(* PLC project Tc3_EventLogger.ipArguments Demo, tc3-libraries-kb TwinCAT 3.1 *)
(* stored: creationDateTime 2026-05-11T01:00:00, modificationDateTime 2026-05-11T01:00:00 *)

PROGRAM P_Demo_ipArguments
  VAR
    fbAlarm : FB_TcAlarm;  (* alarm 实例（已 Create） *)
    ipArgs : I_TcArguments;  (* 参数接口 *)
    sMotorName : STRING := 'M-01';  (* 电机名 *)
    rTemperature : REAL := 95.5;  (* 当前温度 *)
    bAddArgs : BOOL := FALSE;  (* 上升沿触发 *)
    bAddArgsPrev : BOOL;  (* 边沿检测 *)
  END_VAR

// =============================================================================
// 场景：给即将 Raise 的 alarm 附加电机名 + 当前温度两个参数
// 价值：文本占位符自动填充，多语言报警一次代码完成
// 验证：登录后写 bAddArgs := TRUE，触发一次 Add；再 Raise；用 RequestEventText 取回事件文本应包含参数
// 验证步骤：
//   1. 右键 PLC 项目 → Import PLCopenXML → 选本文件
//   2. 引用 Tc3_EventLogger（System → References → Add library）
//   3. 编译 → 登录 → 运行；按 verify 注释里给出的在线写值操作
// =============================================================================

// Raise 之前给 alarm 添加两个参数：电机名 + 温度
IF bAddArgs AND NOT bAddArgsPrev THEN
    ipArgs := fbAlarm.ipArguments;     // 取 getter
    IF ipArgs &lt;&gt; 0 THEN
        ipArgs.AddString(sValue := sMotorName);
        ipArgs.AddReal(fValue := rTemperature);
    END_IF;
END_IF;
bAddArgsPrev := bAddArgs;
END_PROGRAM
